KUKA KRL program: dai_data_library.src, dai_data_library.dat

--- dai_data_library.src ---
&ACCESS RV2
&REL 124
&COMMENT daimler_data_library
&PARAM DISKPATH = KRC:\R1\DAI
&PARAM version = 2.1.1
DEF dai_data_library( )
; Ausgabe der Lade-Meldung....ohne Msg_library weil hier noch nicht geladen
decl KrlMsg_t loadmessage
decl KrlMsgPar_t LoadPar[3]
decl KrlMsgOpt_t loadoptions
decl int handle
loadmessage={modul[] "DAI_MSG_LIB",NR 15,msg_txt[] "DAI_MSG_L4"}
handle=Set_KrlMsg(#notify,loadmessage,LoadPar[],loadoptions)
END

;
;Alle Funktionen fuer die Visu-Signale
;all functions belong to the visu-bits
;
;FOLD VISU

;
; Hauptfunktion fuer die Visusignale
; MainFunction to send the visu-signals
;
GLOBAl DEF Send_Visu_Data()
	; Visu-Signale Senden
 	Visu_Signals()
END

;
;Funktion um die Bits je nach Einstellung zu senden
;
;
DEF Visu_Signals()
 INT iCounter
 INT Number
 CHAR Akt_Shortcut[5]

; Alle fuenf Felder durchlaufen
 FOR iCounter=1 TO 5 STEP 1

    ; Abfrage ob ueberhaupt aktiv ist
   SWITCH Tech_Visu[iCounter].IsActive
		CASE #YES
			; aktuellen Techkueruzel holen
         Akt_Shortcut[]=Tech_Visu[iCounter].TechShortcut[]

			; Arrayposition herausfinden#
         Number = Find_Number(Akt_Shortcut[])

          ; Abfrage ob die Funktion "0" zurueckgegeben hat
          ; --> Kuerzel nicht gefunden
         If (Number == 0) then
          msg_show("DAI_MSG_LIB", #quit, 1, "CTRL_MSG71")
          return
         Endif

			; jetzt werden die Bits gesendet
         Send_Visu_Bits(Tech_Array[Number],iCounter)

		CASE #NO
         SWITCH iCounter
				CASE 1
					Signal_Tech_A_ID = 0
					Signal_Tech_A_DATA = 0
				CASE 2
					Signal_Tech_B_ID = 0
					Signal_Tech_B_DATA = 0
				CASE 3
					Signal_Tech_C_ID = 0
					Signal_Tech_C_DATA = 0
				CASE 4
					Signal_Tech_D_ID = 0
					Signal_Tech_D_DATA = 0
				CASE 5
					Signal_Tech_E_ID = 0
					Signal_Tech_E_DATA = 0
				DEFAULT
					msg_show("DAI_MSG_LIB", #dialog, 1, "CTRL_MSG71")
			ENDSWITCH
		DEFAULT
			msg_show("DAI_MSG_LIB", #quit, 1, "CTRL_MSG70")
	ENDSWITCH
 ENDFOR

END

;
; Unterfunktion die die einzelne Bits sendet
; Subroutine to send the several bits
;
DEF Send_Visu_Bits (Act_Tech:IN,Block:IN)
INT Counter, Block, Offset
Decl Technology Act_tech



    ; Verschiebung der Bloecke berechnen auf Basis der aktuellen Nummer (3553-->Start_Visu)
    Offset = ((Block - 1) * 24) + Start_Visu + 8

		IF Varstate("Act_Tech.Nr1") <> #DECLARED THEN
			SWITCH ACT_Tech.Nr1.Typ
				CASE #INP
               $OUT[0 + Offset] = $IN[Act_Tech.Nr1.Number]
				CASE #OUTP
					$OUT[0 + Offset] = $OUT[Act_Tech.Nr1.Number]
				DEFAULT
					msg_param(1,,Block)
					msg_show("DAI_MSG_LIB", #quit, 1, "CTRL_MSG72")
			ENDSWITCH
		ENDIF
		IF Varstate("Act_Tech.Nr2") <> #DECLARED THEN
			SWITCH ACT_Tech.Nr2.Typ
				CASE #INP
					$OUT[1 + Offset] = $IN[Act_Tech.Nr2.Number]
				CASE #OUTP
					$OUT[1 + Offset] = $OUT[Act_Tech.Nr2.Number]
				DEFAULT
					msg_param(1,,Block)
					msg_show("DAI_MSG_LIB", #quit, 1, "CTRL_MSG73")
			ENDSWITCH
		ENDIF
		IF Varstate("Act_Tech.Nr3") <> #DECLARED THEN
			SWITCH ACT_Tech.Nr3.Typ
				CASE #INP
					$OUT[2 + Offset] = $IN[Act_Tech.Nr3.Number]
				CASE #OUTP
					$OUT[2 + Offset] = $OUT[Act_Tech.Nr3.Number]
				DEFAULT
					msg_param(1,,Block)
					msg_show("DAI_MSG_LIB", #quit, 1, "CTRL_MSG74")
			ENDSWITCH
		ENDIF
		IF Varstate("Act_Tech.Nr4") <> #DECLARED THEN
			SWITCH ACT_Tech.Nr4.Typ
				CASE #INP
					$OUT[3 + Offset] = $IN[Act_Tech.Nr4.Number]
				CASE #OUTP
					$OUT[3 + Offset] = $OUT[Act_Tech.Nr4.Number]
				DEFAULT
					msg_param(1,,Block)
					msg_show("DAI_MSG_LIB", #quit, 1, "CTRL_MSG75")
			ENDSWITCH
		ENDIF
		IF Varstate("Act_Tech.Nr5") <> #DECLARED THEN
			SWITCH ACT_Tech.Nr5.Typ
				CASE #INP
					$OUT[4 + Offset] = $IN[Act_Tech.Nr5.Number]
				CASE #OUTP
					$OUT[4 + Offset] = $OUT[Act_Tech.Nr5.Number]
				DEFAULT
					msg_param(1,,Block)
					msg_show("DAI_MSG_LIB", #quit, 1, "CTRL_MSG76")
			ENDSWITCH
		ENDIF
		IF Varstate("Act_Tech.Nr6") <> #DECLARED THEN
			SWITCH ACT_Tech.Nr6.Typ
				CASE #INP
					$OUT[5 + Offset] = $IN[Act_Tech.Nr6.Number]
				CASE #OUTP
					$OUT[5 + Offset] = $OUT[Act_Tech.Nr6.Number]
				DEFAULT
					msg_param(1,,Block)
					msg_show("DAI_MSG_LIB", #quit, 1, "CTRL_MSG77")
			ENDSWITCH
		ENDIF
		IF Varstate("Act_Tech.Nr7") <> #DECLARED THEN
			SWITCH ACT_Tech.Nr7.Typ
				CASE #INP
					$OUT[6 + Offset] = $IN[Act_Tech.Nr7.Number]
				CASE #OUTP
					$OUT[6 + Offset] = $OUT[Act_Tech.Nr7.Number]
				DEFAULT
					msg_param(1,,Block)
					msg_show("DAI_MSG_LIB", #quit, 1, "CTRL_MSG78")
			ENDSWITCH
		ENDIF
		IF Varstate("Act_Tech.Nr8") <> #DECLARED THEN
			SWITCH ACT_Tech.Nr8.Typ
				CASE #INP
					$OUT[7 + Offset] = $IN[Act_Tech.Nr8.Number]
				CASE #OUTP
					$OUT[7 + Offset] = $OUT[Act_Tech.Nr8.Number]
				DEFAULT
					msg_param(1,,Block)
					msg_show("DAI_MSG_LIB", #quit, 1, "CTRL_MSG79")
			ENDSWITCH
		ENDIF
		IF Varstate("Act_Tech.Nr9") <> #DECLARED THEN
			SWITCH ACT_Tech.Nr9.Typ
				CASE #INP
					$OUT[8 + Offset] = $IN[Act_Tech.Nr9.Number]
				CASE #OUTP
					$OUT[8 + Offset] = $OUT[Act_Tech.Nr9.Number]
				DEFAULT
					msg_param(1,,Block)
					msg_show("DAI_MSG_LIB", #quit, 1, "CTRL_MSG80")
			ENDSWITCH
		ENDIF
		IF Varstate("Act_Tech.Nr10") <> #DECLARED THEN
			SWITCH ACT_Tech.Nr10.Typ
				CASE #INP
					$OUT[9 + Offset] = $IN[Act_Tech.Nr10.Number]
				CASE #OUTP
					$OUT[9 + Offset] = $OUT[Act_Tech.Nr10.Number]
				DEFAULT
					msg_param(1,,Block)
					msg_show("DAI_MSG_LIB", #quit, 1, "CTRL_MSG81")
			ENDSWITCH
		ENDIF
		IF Varstate("Act_Tech.Nr11") <> #DECLARED THEN
			SWITCH ACT_Tech.Nr11.Typ
				CASE #INP
					$OUT[10 + Offset] = $IN[Act_Tech.Nr11.Number]
				CASE #OUTP
					$OUT[10 + Offset] = $OUT[Act_Tech.Nr11.Number]
				DEFAULT
					msg_param(1,,Block)
					msg_show("DAI_MSG_LIB", #quit, 1, "CTRL_MSG82")
			ENDSWITCH
		ENDIF
		IF Varstate("Act_Tech.Nr12") <> #DECLARED THEN
			SWITCH ACT_Tech.Nr12.Typ
				CASE #INP
					$OUT[11 + Offset] = $IN[Act_Tech.Nr12.Number]
				CASE #OUTP
					$OUT[11 + Offset] = $OUT[Act_Tech.Nr12.Number]
				DEFAULT
					msg_param(1,,Block)
					msg_show("DAI_MSG_LIB", #quit, 1, "CTRL_MSG83")
			ENDSWITCH
		ENDIF
		IF Varstate("Act_Tech.Nr13") <> #DECLARED THEN
			SWITCH ACT_Tech.Nr13.Typ
				CASE #INP
					$OUT[12 + Offset] = $IN[Act_Tech.Nr13.Number]
				CASE #OUTP
					$OUT[12 + Offset] = $OUT[Act_Tech.Nr13.Number]
				DEFAULT
					msg_param(1,,Block)
					msg_show("DAI_MSG_LIB", #quit, 1, "CTRL_MSG84")
			ENDSWITCH
		ENDIF
		IF Varstate("Act_Tech.Nr14") <> #DECLARED THEN
			SWITCH ACT_Tech.Nr14.Typ
				CASE #INP
					$OUT[13 + Offset] = $IN[Act_Tech.Nr14.Number]
				CASE #OUTP
					$OUT[13 + Offset] = $OUT[Act_Tech.Nr14.Number]
				DEFAULT
					msg_param(1,,Block)
					msg_show("DAI_MSG_LIB", #quit, 1, "CTRL_MSG85")
			ENDSWITCH
		ENDIF
		IF Varstate("Act_Tech.Nr15") <> #DECLARED THEN
			SWITCH ACT_Tech.Nr15.Typ
				CASE #INP
					$OUT[14 + Offset] = $IN[Act_Tech.Nr15.Number]
				CASE #OUTP
					$OUT[14 + Offset] = $OUT[Act_Tech.Nr15.Number]
				DEFAULT
					msg_param(1,,Block)
					msg_show("DAI_MSG_LIB", #quit, 1, "CTRL_MSG86")
			ENDSWITCH
		ENDIF
		IF Varstate("Act_Tech.Nr16") <> #DECLARED THEN
			SWITCH ACT_Tech.Nr16.Typ
				CASE #INP
					$OUT[15 + Offset] = $IN[Act_Tech.Nr16.Number]
				CASE #OUTP
					$OUT[15 + Offset] = $OUT[Act_Tech.Nr16.Number]
				DEFAULT
					msg_param(1,,Block)
					msg_show("DAI_MSG_LIB", #quit, 1, "CTRL_MSG87")
			ENDSWITCH
		ENDIF

  		;Tech-kennung rueberschieben
		SWITCH Block
		CASE 1
			Signal_Tech_A_ID = ACT_Tech.Kennung
		CASE 2
			Signal_Tech_B_ID = ACT_Tech.Kennung
		CASE 3
			Signal_Tech_C_ID = ACT_Tech.Kennung
		CASE 4
			Signal_Tech_D_ID = ACT_Tech.Kennung
		CASE 5
			Signal_Tech_E_ID = ACT_Tech.Kennung
		DEFAULT
			msg_show("DAI_MSG_LIB", #quit, 1, "CTRL_MSG71")
		ENDSWITCH
END

;
; Unterfunktion: Findet Nummer in dem Array mit dem String wo eingetragen worden isz
; Subroutine to find then number in the Array with the string
;
DEFFCT INT Find_Number (TechShortCutIn[]:IN)
CHAR TechShortCutIn[]
INT Counter
BOOL  bResult

	FOR Counter = 1 TO MAX_TECH STEP 1
      SWITCH Tech_Array[Counter].IsActive
			Case #YES
				IF StrComp(Tech_Array[Counter].TechShortCut[],TechShortCutIn[],#NOT_CASE_SENS) THEN
					return Counter
				ENDIF
			CASE #NO
				; nichts machen
			DEFAULT
				msg_show("DAI_MSG_LIB", #quit, 1, "CTRL_MSG71")
		ENDSWITCH
	ENDFOR

      ; Funktion gibt 0 zurueck wenn die Technologie nicht gefunden wurde
	return 0

ENDFCT

;ENDFOLD


;
;Alle Funktion fuer RDS
;all functions belongs RDS
;
;FOLD RDS


GLOBAL DEF Send_RDS_Data()

; Daten die von der SPS kommen ruerberkopieren auf die einzelnen Bereiche

; 0. Bereich [Byte 480]
O_RDS_0_1 = I_RDS_1
O_RDS_0_2 = I_RDS_2
O_RDS_0_3 = I_RDS_3
O_RDS_0_4 = I_RDS_4
O_RDS_0_5 = I_RDS_5

; 1. Bereich [Byte 600]
O_RDS_1_1 = I_RDS_1
O_RDS_1_2 = I_RDS_2
O_RDS_1_3 = I_RDS_3
O_RDS_1_4 = I_RDS_4
O_RDS_1_5 = I_RDS_5
; 2. Bereich [Byte 620]
O_RDS_2_1 = I_RDS_1
O_RDS_2_2 = I_RDS_2
O_RDS_2_3 = I_RDS_3
O_RDS_2_4 = I_RDS_4
O_RDS_2_5 = I_RDS_5
; 3. Bereich [Byte 640]
O_RDS_3_1 = I_RDS_1
O_RDS_3_2 = I_RDS_2
O_RDS_3_3 = I_RDS_3
O_RDS_3_4 = I_RDS_4
O_RDS_3_5 = I_RDS_5
; 4. Bereich [Byte 660]
O_RDS_4_1 = I_RDS_1
O_RDS_4_2 = I_RDS_2
O_RDS_4_3 = I_RDS_3
O_RDS_4_4 = I_RDS_4
O_RDS_4_5 = I_RDS_5
; 5. Bereich [Byte 680]
O_RDS_5_1 = I_RDS_1
O_RDS_5_2 = I_RDS_2
O_RDS_5_3 = I_RDS_3
O_RDS_5_4 = I_RDS_4
O_RDS_5_5 = I_RDS_5
; 6. Bereich [Byte 700]
O_RDS_6_1 = I_RDS_1
O_RDS_6_2 = I_RDS_2
O_RDS_6_3 = I_RDS_3
O_RDS_6_4 = I_RDS_4
O_RDS_6_5 = I_RDS_5
; 7. Bereich [Byte 720]
O_RDS_7_1 = I_RDS_1
O_RDS_7_2 = I_RDS_2
O_RDS_7_3 = I_RDS_3
O_RDS_7_4 = I_RDS_4
O_RDS_7_5 = I_RDS_5
; 8. Bereich [Byte 740]
O_RDS_8_1 = I_RDS_1
O_RDS_8_2 = I_RDS_2
O_RDS_8_3 = I_RDS_3
O_RDS_8_4 = I_RDS_4
O_RDS_8_5 = I_RDS_5
; 9. Bereich [Byte 760]
O_RDS_9_1 = I_RDS_1
O_RDS_9_2 = I_RDS_2
O_RDS_9_3 = I_RDS_3
O_RDS_9_4 = I_RDS_4
O_RDS_9_5 = I_RDS_5
; 10. Bereich [Byte 780]
O_RDS_10_1 = I_RDS_1
O_RDS_10_2 = I_RDS_2
O_RDS_10_3 = I_RDS_3
O_RDS_10_4 = I_RDS_4
O_RDS_10_5 = I_RDS_5
; 11. Bereich [Byte 800]
O_RDS_11_1 = I_RDS_1
O_RDS_11_2 = I_RDS_2
O_RDS_11_3 = I_RDS_3
O_RDS_11_4 = I_RDS_4
O_RDS_11_5 = I_RDS_5
END

;ENDFOLD


;
;Alle Funktion fuer PLUS
;all functions belongs PLUS
;
;FOLD PLUS

; Globale Funktion für die PLUS-Anbindung
; global function for PLUS-coupling
GLOBAL DEF  PlusData(PLUS_CMD: IN,PLUS_Data: IN)
    DECL en_PlusData PLUS_CMD
    DECL T_PlusData PLUS_Data

    switch PLUS_CMD
    case #PLUS_Init
        PlusData_Init()
    case #PLUS_Fill
        PlusData_Fill(PLUS_Data)
    case #PLUS_Send
        PlusData_Send()
    default
    ;
    endswitch

END

; Funktion zum Initialisieren der Gesamten PLUS-Funktion
; Initialize the complete PLUS-function
DEF PlusData_Init()
    Result = true
    time = 1

    ; Abfrage ob Uerbtragung das letzte Mal erfolgreich
    IF  bPLUSSend THEN        ; Wenn ich was gesendet habe
      IF NOT $IN[IO_AzykHndshkPLC]  THEN    ; und keine erfolgreiche Rückmeldung habe
         Msg_Show("DAI_MSG_LIB",#notify,10,"QD_DLG_MSG10") ;Letzte Q-Daten wurden von SPS nicht gelesen
      ENDIF
      bPLUSSend = FALSE ; Merker wieder zuruecksetzen
    ENDIF

    ; Request an SPS nochmals wegnehmen falls es beim letzten Senden einen Fehler gab
    $OUT[IO_AzykHndshkPLC] = FALSE

    ; Sendebuffer leer machen
    wait for StrClear(SendBuffer[])

    ; Temp Datenspeicher loeschen
    TempQTelegram.QAussageArt[] = "    " ;4Zeichen
    TempQTelegram.qcodierung[] = "    " ;4Zeichen
    TempQTelegram.qident[] = "            " ;12 Zeichen

    ; Array leer machen & Zaehler zuruecksetzebn
    FOR SpotNr=1 TO Max_PlusData
    	  QualTelegram[SpotNr].QAussageArt[] = "    "
        QualTelegram[SpotNr].QIdent[] = 	"            "
        QualTelegram[SpotNr].QCodierung[] = "    "
    ENDFOR
    SpotNr = 1

     ; Azyklischen Dienst initialisieren
     AzykHndl = 0
     WModus = #ASYNC
     offset = 0
     COPEN(:LD_EXT_OBJ1,AzykHndl) ; Link auf External Object in machine.dat
END

; Funktion fuer die Techpakete um die Punkt zu fuellen
; function for the techpakets to fill the PLUS-array
DEF PlusData_Fill(PLUS_Data :IN)
   DECL T_PlusData PLUS_Data
   ;Check ob noch PLatz im Array
   IF (SpotNr > Max_PlusData) THEN
		Msg_Show("DAI_MSG_LIB",#quit,10,"QD_DLG_MSG11")
		HALT
   ENDIF

   ; Daten werden ins Array kopiert

   ; Punktnummer wird reinkopiert
   wait for   StrCopy(QualTelegram[SpotNr].QIdent[],PLUS_Data.QIdent[])
   wait for   StrCopy(QualTelegram[SpotNr].QAussageArt[],PLUS_Data.QAussageArt[])
   wait for   StrCopy(QualTelegram[SpotNr].QCodierung[],PLUS_Data.QCodierung[])

   ; Punktzaehler wir hochgezaehlt
   SpotNr = SpotNr + 1

   ; temporaere Daten loeschen
   PLUS_Data.QAussageArt[] = "    " ;4Zeichen
   PLUS_Data.qcodierung[] = "    " ;4Zeichen
   PLUS_Data.qident[] = "            " ;12 Zeichen
   TempQTelegram.QAussageArt[] = "    " ;4Zeichen
   TempQTelegram.qcodierung[] = "    " ;4Zeichen
   TempQTelegram.qident[] = "            " ;12 Zeichen



END


; Funktion um die Daten azyklisch zu senden
; function to send the data
DEF PlusData_Send()
DECL INT iLauf



IF (SpotNr > 1) AND (bPLUSActiv)  THEN

      ; IO-Request an SPS schicken
      $OUT[IO_AzykHndshkPLC] = TRUE

      IF AzykHndl > 0 then


         ; INIT-Telegramm von SPS empfangen
         RModus = #ABS
         CREAD(AzykHndl,WState,RModus, TimeOut, offset,"%r",SendBuffer[])

         IF (WState.Ret1 == #Data_End) then
            wait sec 0.2
            offset = 0

            ; Daten aus dem Requesttelegramm rauslesen
           	CAST_FROM(SendBuffer[],offset,cmdid)
           	CAST_FROM(SendBuffer[],offset,cmdl)
           	CAST_FROM(SendBuffer[],offset,tid)
           	CAST_FROM(SendBuffer[],offset,aid)
           	CAST_FROM(SendBuffer[],offset,slot)
           	CAST_FROM(SendBuffer[],offset,sslot)
           	CAST_FROM(SendBuffer[],offset,idx)
          	CAST_FROM(SendBuffer[],offset,cdl)

            ; ID 3 --> Requesttelegramm
            IF (cmdid == 3) THEN
            	offset = 0
           		CAST_TO(SendBuffer[],offset,cmdid)
               cmdl = 2028 ; 2000Bytes Nutzdaten  + 28Bytes Header
           		CAST_TO(SendBuffer[],offset,cmdl)
           		CAST_TO(SendBuffer[],offset,tid)
           		CAST_TO(SendBuffer[],offset,aid)
           		CAST_TO(SendBuffer[],offset,slot)
           		CAST_TO(SendBuffer[],offset,sslot)
           		CAST_TO(SendBuffer[],offset,idx)
           		errc = 0
           		CAST_TO(SendBuffer[],offset,errc)
           		CAST_TO(SendBuffer[],offset,cdl)

               ; Jetzt die einzelnen Punkte rausschreiben
               FOR iLauf=1 TO Max_PlusData
               	 ;GLOBAL STRUC T_PlusData CHAR QAussageArt[4], CHAR QIdent[12],CHAR QCodierung[4]
               	CAST_TO(SendBuffer[],offset,QualTelegram[iLauf].QAussageArt[])
                  CAST_TO(SendBuffer[],offset,QualTelegram[iLauf].QIdent[])
                  CAST_TO(SendBuffer[],offset,QualTelegram[iLauf].QCodierung[])
               ENDFOR

               ; Jetzt das eigentliche Paket wegschicken
               CWrite(AzykHndl,WState,WModus,"%1.2036r",SendBuffer[])
            ENDIF
         ENDIF
      ENDIF
      wait sec 0.5

      ;IO-Request an SPS wegnehmen
      $OUT[IO_AzykHndshkPLC] = FALSE




ENDIF
END

;ENDFOLD

--- dai_data_library.dat ---
&ACCESS RV2
&REL 124
&COMMENT daimler_data_library
&PARAM DISKPATH = KRC:\R1\DAI
&PARAM version = 2.1.1
DEFDAT  dai_data_library PUBLIC


;FOLD VISU --don't touch--

; Daten
GLOBAL ENUM IO_TYP INP,OUTP
GLOBAL ENUM YesNo No,YES
GLOBAL STRUC Tech CHAR TechShortcut[5],YesNo IsActive
GLOBAL STRUC DigitalIO INT Number,IO_TYP Typ
GLOBAL STRUC Technology YesNo IsActive,CHAR TechShortCut[5],INT Kennung,DigitalIO Nr1,DigitalIO Nr2,DigitalIO Nr3,DigitalIO Nr4,DigitalIO Nr5,DigitalIO Nr6,DigitalIO Nr7,DigitalIO Nr8,DigitalIO Nr9,DigitalIO Nr10,DigitalIO Nr11,DigitalIO Nr12,DigitalIO Nr13,DigitalIO Nr14,DigitalIO Nr15,DigitalIO Nr16
DECL CONST INT Start_Visu=3553
;feste Signalvereinbarungen, da dies aktuell noch nicht dynamisch gemacht werden kann
;und die dynamische Funktion uerbs Ziel hinausgeschossen waere
SIGNAL Signal_Tech_A_ID $OUT[3553]  TO $OUT[3560]
SIGNAL Signal_Tech_A_Data $OUT[3561]  TO $OUT[3576]

SIGNAL Signal_Tech_B_ID $OUT[3577]  TO $OUT[3584]
SIGNAL Signal_Tech_B_Data $OUT[3585]  TO $OUT[3600]

SIGNAL Signal_Tech_C_ID $OUT[3601]  TO $OUT[3608]
SIGNAL Signal_Tech_C_Data $OUT[3609]  TO $OUT[3624]

SIGNAL Signal_Tech_D_ID $OUT[3625]  TO $OUT[3632]
SIGNAL Signal_Tech_D_Data $OUT[3633]  TO $OUT[3648]

SIGNAL Signal_Tech_E_ID $OUT[3649]  TO $OUT[3656]
SIGNAL Signal_Tech_E_Data $OUT[3657]  TO $OUT[3672]

;ENDFOLD

;FOLD RDS --don't touch--

; Maximale Signalelaenge 32bit --> 4 bytes immer
Decl GLOBAL Bool WithRDS=FALSE
;Eingangsbeschreibung der Daten von der SPS auf der Schnittstelle
SIGNAL I_RDS_1 $IN[1026]  TO $IN[1026]
SIGNAL I_RDS_2 $IN[1026]  TO $IN[1026]
SIGNAL I_RDS_3 $IN[1026]  TO $IN[1026]
SIGNAL I_RDS_4 $IN[1026]  TO $IN[1026]
SIGNAL I_RDS_5 $IN[1026]  TO $IN[1026]

; Erste, interne Spiegelung der Daten auf einen Eíngangsbereich
SIGNAL O_RDS_0_1 $OUT[999]  TO $OUT[999]
SIGNAL O_RDS_0_2 $OUT[999]  TO $OUT[999]
SIGNAL O_RDS_0_3 $OUT[999]  TO $OUT[999]
SIGNAL O_RDS_0_4 $OUT[999]  TO $OUT[999]
SIGNAL O_RDS_0_5 $OUT[999]  TO $OUT[999]


; 1. Bereich fürt die Technologien ab Byte 600 (8k-Bereich)
SIGNAL O_RDS_1_1 $OUT[999]  TO $OUT[999]
SIGNAL O_RDS_1_2 $OUT[999]  TO $OUT[999]
SIGNAL O_RDS_1_3 $OUT[999]  TO $OUT[999]
SIGNAL O_RDS_1_4 $OUT[999]  TO $OUT[999]
SIGNAL O_RDS_1_5 $OUT[999]  TO $OUT[999]
; 2. Bereich
SIGNAL O_RDS_2_1 $OUT[999]  TO $OUT[999]
SIGNAL O_RDS_2_2 $OUT[999]  TO $OUT[999]
SIGNAL O_RDS_2_3 $OUT[999]  TO $OUT[999]
SIGNAL O_RDS_2_4 $OUT[999]  TO $OUT[999]
SIGNAL O_RDS_2_5 $OUT[999]  TO $OUT[999]
; 3. Bereich
SIGNAL O_RDS_3_1 $OUT[999]  TO $OUT[999]
SIGNAL O_RDS_3_2 $OUT[999]  TO $OUT[999]
SIGNAL O_RDS_3_3 $OUT[999]  TO $OUT[999]
SIGNAL O_RDS_3_4 $OUT[999]  TO $OUT[999]
SIGNAL O_RDS_3_5 $OUT[999]  TO $OUT[999]
; 4. Bereich
SIGNAL O_RDS_4_1 $OUT[999]  TO $OUT[999]
SIGNAL O_RDS_4_2 $OUT[999]  TO $OUT[999]
SIGNAL O_RDS_4_3 $OUT[999]  TO $OUT[999]
SIGNAL O_RDS_4_4 $OUT[999]  TO $OUT[999]
SIGNAL O_RDS_4_5 $OUT[999]  TO $OUT[999]
; 5. Bereich
SIGNAL O_RDS_5_1 $OUT[999]  TO $OUT[999]
SIGNAL O_RDS_5_2 $OUT[999]  TO $OUT[999]
SIGNAL O_RDS_5_3 $OUT[999]  TO $OUT[999]
SIGNAL O_RDS_5_4 $OUT[999]  TO $OUT[999]
SIGNAL O_RDS_5_5 $OUT[999]  TO $OUT[999]
; 6. Bereich
SIGNAL O_RDS_6_1 $OUT[999]  TO $OUT[999]
SIGNAL O_RDS_6_2 $OUT[999]  TO $OUT[999]
SIGNAL O_RDS_6_3 $OUT[999]  TO $OUT[999]
SIGNAL O_RDS_6_4 $OUT[999]  TO $OUT[999]
SIGNAL O_RDS_6_5 $OUT[999]  TO $OUT[999]
; 7. Bereich
SIGNAL O_RDS_7_1 $OUT[999]  TO $OUT[999]
SIGNAL O_RDS_7_2 $OUT[999]  TO $OUT[999]
SIGNAL O_RDS_7_3 $OUT[999]  TO $OUT[999]
SIGNAL O_RDS_7_4 $OUT[999]  TO $OUT[999]
SIGNAL O_RDS_7_5 $OUT[999]  TO $OUT[999]
; 8. Bereich
SIGNAL O_RDS_8_1 $OUT[999]  TO $OUT[999]
SIGNAL O_RDS_8_2 $OUT[999]  TO $OUT[999]
SIGNAL O_RDS_8_3 $OUT[999]  TO $OUT[999]
SIGNAL O_RDS_8_4 $OUT[999]  TO $OUT[999]
SIGNAL O_RDS_8_5 $OUT[999]  TO $OUT[999]
; 9. Bereich
SIGNAL O_RDS_9_1 $OUT[999]  TO $OUT[999]
SIGNAL O_RDS_9_2 $OUT[999]  TO $OUT[999]
SIGNAL O_RDS_9_3 $OUT[999]  TO $OUT[999]
SIGNAL O_RDS_9_4 $OUT[999]  TO $OUT[999]
SIGNAL O_RDS_9_5 $OUT[999]  TO $OUT[999]
; 10. Bereich
SIGNAL O_RDS_10_1 $OUT[999]  TO $OUT[999]
SIGNAL O_RDS_10_2 $OUT[999]  TO $OUT[999]
SIGNAL O_RDS_10_3 $OUT[999]  TO $OUT[999]
SIGNAL O_RDS_10_4 $OUT[999]  TO $OUT[999]
SIGNAL O_RDS_10_5 $OUT[999]  TO $OUT[999]
; 11. Bereich
SIGNAL O_RDS_11_1 $OUT[999]  TO $OUT[999]
SIGNAL O_RDS_11_2 $OUT[999]  TO $OUT[999]
SIGNAL O_RDS_11_3 $OUT[999]  TO $OUT[999]
SIGNAL O_RDS_11_4 $OUT[999]  TO $OUT[999]
SIGNAL O_RDS_11_5 $OUT[999]  TO $OUT[999]
;ENDFOLD

;FOLD PLUS --don't touch--
GLOBAL ENUM en_PlusData PLUS_Init,PLUS_Fill,PLUS_Send
GLOBAL STRUC T_PlusData CHAR QAussageArt[4], CHAR QIdent[12],CHAR QCodierung[4]

DECL CONST INT Max_PlusData=100
DECL CONST INT IO_AzykHndshkPLC=3227
DECL T_PlusData QualTelegram[200]
DECL GLOBAL T_PlusData TempQTelegram
CHAR SendBuffer[2200]

DECL STATE_T WState
DECL MODUS_T WModus,RModus

DECL INT SpotNr,offset,AzykHndl,Time
DECL REAL TimeOut=5.0
DECL INT cmdid,cmdl,tid,aid,slot,sslot,idx,cdl,errc
DECL BOOL Result
DECL BOOL bPLUSSend = FALSE
DECL CONST BOOL bPLUSActiv = TRUE

;ENDFOLD



;FOLD Technologien

DECL CONST INT Max_Tech=40

DECL GLOBAL Technology Tech_Array[40]
Tech_Array[1]={IsActive #YES,TechShortCut[] "SWP_1",Kennung 1,Nr1 {Number 516,Typ #INP},Nr2 {Number 529,Typ #INP},Nr3 {Number 531,Typ #INP},Nr4 {Number 533,Typ #INP},Nr5 {Number 534,Typ #INP},Nr6 {Number 535,Typ #INP},Nr7 {Number 547,Typ #INP},Nr8 {Number 552,Typ #INP},Nr9 {Number 569,Typ #INP}}
Tech_Array[2]={IsActive #YES,TechShortCut[] "SWP_2",Kennung 2,Nr1 {Number 516,Typ #INP},Nr2 {Number 529,Typ #INP},Nr3 {Number 531,Typ #INP},Nr4 {Number 533,Typ #INP},Nr5 {Number 534,Typ #INP},Nr6 {Number 535,Typ #INP},Nr7 {Number 547,Typ #INP},Nr8 {Number 552,Typ #INP},Nr9 {Number 569,Typ #INP}}
Tech_Array[3]={IsActive #YES,TechShortCut[] "SWB_1",Kennung 3,Nr1 {Number 1153,Typ #INP},Nr2 {Number 1155,Typ #INP},Nr3 {Number 1184,Typ #INP}}
Tech_Array[4]={IsActive #YES,TechShortCut[] "SWB_2",Kennung 4,Nr1 {Number 1153,Typ #INP},Nr2 {Number 1155,Typ #INP},Nr3 {Number 1184,Typ #INP}}
Tech_Array[5]={IsActive #YES,TechShortCut[] "SWM_1",Kennung 5,Nr1 {Number 1892,Typ #INP},Nr2 {Number 1899,Typ #INP},Nr3 {Number 1900,Typ #INP},Nr4 {Number 1901,Typ #INP},Nr5 {Number 1902,Typ #INP}}
Tech_Array[6]={IsActive #YES,TechShortCut[] "SWM_2",Kennung 6,Nr1 {Number 1892,Typ #INP},Nr2 {Number 1899,Typ #INP},Nr3 {Number 1900,Typ #INP},Nr4 {Number 1901,Typ #INP},Nr5 {Number 1902,Typ #INP}}
Tech_Array[7]={IsActive #YES,TechShortCut[] "MNI_1",Kennung 7,Nr1 {Number 2879,Typ #INP},Nr2 {Number 2880,Typ #INP}}
Tech_Array[8]={IsActive #YES,TechShortCut[] "MNI_2",Kennung 8,Nr1 {Number 2879,Typ #INP},Nr2 {Number 2880,Typ #INP}}
Tech_Array[9]={IsActive #YES,TechShortCut[] "KLB_1",Kennung 9,Nr1 {Number 1537,Typ #INP},Nr2 {Number 1538,Typ #INP},Nr3 {Number 1569,Typ #INP},Nr4 {Number 1571,Typ #INP},Nr5 {Number 1601,Typ #INP},Nr6 {Number 1602,Typ #INP},Nr7 {Number 1603,Typ #INP},Nr8 {Number 1604,Typ #INP},Nr9 {Number 1605,Typ #INP},Nr10 {Number 1606,Typ #INP},Nr11 {Number 1607,Typ #INP},Nr12 {Number 1608,Typ #INP},Nr13 {Number 1609,Typ #INP}}
Tech_Array[10]={IsActive #YES,TechShortCut[] "KLB_2",Kennung 10,Nr1 {Number 1665,Typ #INP},Nr2 {Number 1666,Typ #INP},Nr3 {Number 1697,Typ #INP},Nr4 {Number 1699,Typ #INP},Nr5 {Number 1729,Typ #INP},Nr6 {Number 1731,Typ #INP},Nr7 {Number 1732,Typ #INP},Nr8 {Number 1734,Typ #INP}}
Tech_Array[11]={IsActive #YES,TechShortCut[] "KNI_1",Kennung 11,Nr1 {Number 1601,Typ #INP},Nr2 {Number 1602,Typ #INP},Nr3 {Number 1603,Typ #INP},Nr4 {Number 1604,Typ #INP},Nr5 {Number 1605,Typ #INP},Nr6 {Number 1606,Typ #INP},Nr7 {Number 1607,Typ #INP},Nr8 {Number 1608,Typ #INP},Nr9 {Number 1609,Typ #INP},Nr10 {Number 1610,Typ #INP},Nr11 {Number 1611,Typ #INP},Nr12 {Number 1612,Typ #INP},Nr13 {Number 1613,Typ #INP},Nr14 {Number 1614,Typ #OUTP}}
Tech_Array[12]={IsActive #YES,TechShortCut[] "KNI_2",Kennung 12,Nr1 {Number 1729,Typ #INP},Nr2 {Number 1730,Typ #INP},Nr3 {Number 1731,Typ #INP},Nr4 {Number 1732,Typ #INP},Nr5 {Number 1733,Typ #INP},Nr6 {Number 1734,Typ #INP},Nr7 {Number 1735,Typ #INP},Nr8 {Number 1736,Typ #INP},Nr9 {Number 1737,Typ #INP},Nr10 {Number 1738,Typ #INP},Nr11 {Number 1739,Typ #INP},Nr12 {Number 1740,Typ #INP},Nr13 {Number 1741,Typ #INP},Nr14 {Number 1742,Typ #OUTP}}
Tech_Array[13]={IsActive #YES,TechShortCut[] "VSN_1",Kennung 13}
Tech_Array[14]={IsActive #YES,TechShortCut[] "VSN_2",Kennung 14}
Tech_Array[15]={IsActive #YES,TechShortCut[] "HSN_1",Kennung 15,Nr1 {Number 2632,Typ #INP},Nr2 {Number 2634,Typ #INP},Nr3 {Number 2635,Typ #INP},Nr4 {Number 2640,Typ #INP},Nr5 {Number 2646,Typ #INP},Nr6 {Number 2647,Typ #INP},Nr7 {Number 2648,Typ #INP},Nr8 {Number 2657,Typ #INP},Nr9 {Number 2658,Typ #INP},Nr10 {Number 2659,Typ #INP}}
Tech_Array[16]={IsActive #YES,TechShortCut[] "HSN_2",Kennung 16,Nr1 {Number 2632,Typ #INP},Nr2 {Number 2634,Typ #INP},Nr3 {Number 2635,Typ #INP},Nr4 {Number 2640,Typ #INP},Nr5 {Number 2646,Typ #INP},Nr6 {Number 2647,Typ #INP},Nr7 {Number 2648,Typ #INP},Nr8 {Number 2657,Typ #INP},Nr9 {Number 2658,Typ #INP},Nr10 {Number 2659,Typ #INP}}
Tech_Array[17]={IsActive #YES,TechShortCut[] "FZR_1",Kennung 17,Nr1 {Number 1921,Typ #INP},Nr2 {Number 1922,Typ #INP},Nr3 {Number 1923,Typ #INP},Nr4 {Number 1953,Typ #INP},Nr5 {Number 1955,Typ #INP},Nr6 {Number 1921,Typ #OUTP},Nr7 {Number 1929,Typ #OUTP}}
Tech_Array[18]={IsActive #YES,TechShortCut[] "FZR_2",Kennung 18,Nr1 {Number 1921,Typ #INP},Nr2 {Number 1922,Typ #INP},Nr3 {Number 1923,Typ #INP},Nr4 {Number 1953,Typ #INP},Nr5 {Number 1955,Typ #INP},Nr6 {Number 1921,Typ #OUTP},Nr7 {Number 1929,Typ #OUTP}}
Tech_Array[19]={IsActive #YES,TechShortCut[] "IMP_1",Kennung 19,Nr1 {Number 3027,Typ #INP},Nr2 {Number 3028,Typ #INP},Nr3 {Number 3029,Typ #INP},Nr4 {Number 3033,Typ #INP},Nr5 {Number 3038,Typ #INP},Nr6 {Number 3039,Typ #INP},Nr7 {Number 3034,Typ #INP},Nr8 {Number 3035,Typ #INP},Nr9 {Number 3036,Typ #INP}}
Tech_Array[20]={IsActive #YES,TechShortCut[] "IMP_2",Kennung 20,Nr1 {Number 3027,Typ #INP},Nr2 {Number 3028,Typ #INP},Nr3 {Number 3029,Typ #INP},Nr4 {Number 3033,Typ #INP},Nr5 {Number 3038,Typ #INP},Nr6 {Number 3039,Typ #INP},Nr7 {Number 3034,Typ #INP},Nr8 {Number 3035,Typ #INP},Nr9 {Number 3036,Typ #INP}}
Tech_Array[21]={IsActive #YES,TechShortCut[] "SRF_1",Kennung 21,Nr1 {Number 2401,Typ #INP},Nr2 {Number 2402,Typ #INP},Nr3 {Number 2403,Typ #INP},Nr4 {Number 2404,Typ #INP},Nr5 {Number 2405,Typ #INP},Nr6 {Number 2406,Typ #INP},Nr7 {Number 2407,Typ #INP},Nr8 {Number 2408,Typ #INP}}
Tech_Array[22]={IsActive #YES,TechShortCut[] "SRF_2",Kennung 22,Nr1 {Number 2401,Typ #INP},Nr2 {Number 2402,Typ #INP},Nr3 {Number 2403,Typ #INP},Nr4 {Number 2404,Typ #INP},Nr5 {Number 2405,Typ #INP},Nr6 {Number 2406,Typ #INP},Nr7 {Number 2407,Typ #INP},Nr8 {Number 2408,Typ #INP}}
Tech_Array[23]={IsActive #YES,TechShortCut[] "CLS_1",Kennung 23,Nr1 {Number 1409,Typ #INP},Nr2 {Number 1411,Typ #INP},Nr3 {Number 1419,Typ #INP},Nr4 {Number 1425,Typ #INP},Nr5 {Number 1426,Typ #INP},Nr6 {Number 1430,Typ #INP},Nr7 {Number 1432,Typ #INP},Nr8 {Number 1433,Typ #INP},Nr9 {Number 1438,Typ #INP},Nr10 {Number 1435,Typ #INP},Nr11 {Number 1437,Typ #INP}}
Tech_Array[24]={IsActive #YES,TechShortCut[] "CLS_2",Kennung 24,Nr1 {Number 1473,Typ #INP},Nr2 {Number 1475,Typ #INP},Nr3 {Number 1483,Typ #INP},Nr4 {Number 1489,Typ #INP},Nr5 {Number 1490,Typ #INP},Nr6 {Number 1494,Typ #INP},Nr7 {Number 1496,Typ #INP},Nr8 {Number 1497,Typ #INP},Nr9 {Number 1502,Typ #INP},Nr10 {Number 1499,Typ #INP},Nr11 {Number 1501,Typ #INP}}
Tech_Array[25]={IsActive #YES,TechShortCut[] "CF__1",Kennung 25}
Tech_Array[26]={IsActive #YES,TechShortCut[] "CF__2",Kennung 26}
Tech_Array[27]={IsActive #YES,TechShortCut[] "QDL_1",Kennung 27,Nr1 {Number 2865,Typ #INP},Nr2 {Number 2867,Typ #INP},Nr3 {Number 2871,Typ #INP},Nr4 {Number 2872,Typ #INP},Nr5 {Number 2873,Typ #INP},Nr6 {Number 2874,Typ #INP}}
Tech_Array[28]={IsActive #YES,TechShortCut[] "QDL_2",Kennung 28,Nr1 {Number 2865,Typ #INP},Nr2 {Number 2867,Typ #INP},Nr3 {Number 2871,Typ #INP},Nr4 {Number 2872,Typ #INP},Nr5 {Number 2873,Typ #INP},Nr6 {Number 2874,Typ #INP}}
Tech_Array[29]={IsActive #YES,TechShortCut[] "TAR_1",Kennung 29,Nr1 {Number 2250,Typ #INP},Nr2 {Number 2251,Typ #INP}}
Tech_Array[30]={IsActive #YES,TechShortCut[] "TAR_2",Kennung 30,Nr1 {Number 2250,Typ #INP},Nr2 {Number 2251,Typ #INP}}
Tech_Array[31]={IsActive #No}
Tech_Array[32]={IsActive #No}
Tech_Array[33]={IsActive #No}
Tech_Array[34]={IsActive #No}
Tech_Array[35]={IsActive #No}
Tech_Array[36]={IsActive #No}
Tech_Array[37]={IsActive #No}
Tech_Array[38]={IsActive #No}
Tech_Array[39]={IsActive #No}
Tech_Array[40]={IsActive #No}
;ENDFOLD




ENDDAT
